INTERFACE I_AsyncResponseHeaderAccessor

METHOD PUBLIC TryGetResponseIdFromRequest : BOOL
VAR_INPUT
	Request : I_Request;
	Destination : ANY;
END_VAR
END_METHOD

METHOD PUBLIC TryGetSessionIdFromRequest : BOOL
VAR_INPUT
	Request : I_Request;
	Destination : REFERENCE TO T_MAXSTRING;
END_VAR
END_METHOD

METHOD PUBLIC TryGetSessionIdFromResponse : BOOL
VAR_INPUT
	Response : I_ServerResponse;
	Destination : ANY;
END_VAR
END_METHOD

END_INTERFACE

(* stored: Version 1.1.0.1, ProductVersion 3.1.4024.12
   Itf I_AsyncResponseHeaderAccessor: Id {f6f392da-89e0-0f59-09ca-702f62293862}
   Method TryGetResponseIdFromRequest: Id {cd1dbc8e-de55-0a1e-1dea-0c99145cdb7b}
   Method TryGetSessionIdFromRequest: Id {ceb58ee4-e2c1-0445-1490-e34c6b55beca}
   Method TryGetSessionIdFromResponse: Id {1e289d15-3bec-0069-2806-9b18d052ed13} *)
